# EPICS substitutions: iocBoot/iocHindsXray/pid_slow.substitutions
file "$(STD)/db/pid_control.db"
{
pattern
{P,            PID,        INP,             OUT,               LOPR,  HOPR,  DRVL,  DRVH,  PREC,   KP,  KI,   KD,  SCAN}
{HindsXray:,  PID1, HindsXray:ETC:Ti1, HindsXray:USB2408:Ao1,   0,    100,     0,    5,     3,     0.2,  3.,   0.,  ".1 second"}
}
